// TwinCAT 3 PLC project OEAMTC_WienWest
// ProgramVersion: 3.1.4023.0
// libraries:
//   EfficientIO Communicator, * (EfficientIO)
//   Lynus Energy Basic, * (Lynus AG)
//   Lynus Persistent Data V1, * (Lynus AG)
//   Lynus Standards, * (Lynus AG)
//   Tc2_ModbusRTU, * (Beckhoff Automation GmbH)
//   Tc2_SerialCom, * (Beckhoff Automation GmbH)
//   Tc2_Standard, * (Beckhoff Automation GmbH)
//   Tc2_System, * (Beckhoff Automation GmbH)
//   Tc2_Utilities, * (Beckhoff Automation GmbH)
//   Tc3_Module, * (Beckhoff Automation GmbH)
// project tree:
//   DUTs/ ModbusRTURequest.TcDUT
//   / FastTask.TcTTO, MiddleTask.TcTTO, SlowTask.TcTTO
//   FB/ F_Convert_Reg_to_Real.TcPOU, MODBUS_RTU_v0.TcPOU
//   POUs/ prgComEffIO.TcPOU, prgMain.TcPOU, prgPersistent.TcPOU, prgPV.TcPOU (excluded from build), prgRWEffIO.TcPOU, prgVarEffIO.TcPOU
// real-time tasks:
//   TASK MiddleTask: cycle T#10ms, priority 20, ADS port 350
//   TASK SlowTask: cycle T#20ms, priority 21, ADS port 351
//   TASK FastTask: cycle T#5ms, priority 19, ADS port 352
// I/O:
//   DEVICE Device 1 (Beckhoff CCAT)
//   DEVICE Device 2 (CX-BK)
//     Box 1 (CX-BK)
// variable links:
//   OEAMTC_WienWest/OEAMTC_WienWest Instance <-> Device 2 (CX-BK)/Box 1 (CX-BK)
//     FastTask Inputs/MODBUS_RTU_v0.fbModbusRtuMaster_KL6x22B.InData/D <-> Term 2 (KL6041)/Channel 1/Data In 0
//     FastTask Inputs/MODBUS_RTU_v0.fbModbusRtuMaster_KL6x22B.InData/D @bit {8..168 step 8} <-> Term 2 (KL6041)/Channel 1/Data In {1..21}  (21 links)
//     FastTask Inputs/MODBUS_RTU_v0.fbModbusRtuMaster_KL6x22B.InData/Status <-> Term 2 (KL6041)/Channel 1/State
//     FastTask Inputs/prgMain.fbKBusState.uiKBusState_OUT <-> Inputs/State
//     FastTask Outputs/MODBUS_RTU_v0.fbModbusRtuMaster_KL6x22B.OutData/Ctrl <-> Term 2 (KL6041)/Channel 1/Ctrl
//     FastTask Outputs/MODBUS_RTU_v0.fbModbusRtuMaster_KL6x22B.OutData/D <-> Term 2 (KL6041)/Channel 1/Data Out 0
//     FastTask Outputs/MODBUS_RTU_v0.fbModbusRtuMaster_KL6x22B.OutData/D @bit {8..168 step 8} <-> Term 2 (KL6041)/Channel 1/Data Out {1..21}  (21 links)

CONFIGURATION OEAMTC_WienWest
    RESOURCE PLC ON TwinCAT3
        TASK FastTask(INTERVAL := T#5ms, PRIORITY := 19);
        TASK MiddleTask(INTERVAL := T#10ms, PRIORITY := 20);
        TASK SlowTask(INTERVAL := T#20ms, PRIORITY := 21);
        PROGRAM prgRWEffIO WITH FastTask : prgRWEffIO;
        PROGRAM prgVarEffIO WITH FastTask : prgVarEffIO;
        PROGRAM prgMain WITH FastTask : prgMain;
        PROGRAM prgPersistent WITH MiddleTask : prgPersistent;
        PROGRAM prgComEffIO WITH SlowTask : prgComEffIO;
    END_RESOURCE
END_CONFIGURATION

// ---- DUTs/ModbusRTURequest.TcDUT
TYPE ModbusRTURequest :
STRUCT
	byteClientSlaveID	:BYTE;
	uintStartAddress	:UINT;
	uintNoOfWords		:UINT;
	mError				:BOOL;
	udintErrorID		:MODBUS_ERRORS;
	udintBytesReceived	:UDINT;
	timerErrorTimer		:TON;
	timerOKTimer		:TON;
	wArrayReceiveBuffer	:ARRAY[0..130] OF WORD;
	udintReceiveBufferAddress	:UDINT;
	strErrorMessage		:STRING(50);
	udintCommErrorCounter		:UDINT;
	udintCommSuccessCounter		:UDINT;
	timeTimeForRequest	:TIME;
	mRequestActive		:BOOL;
	intDeviceClass		:INT;
	intDeviceNumber		:INT;
END_STRUCT
END_TYPE

// ---- POUs/prgRWEffIO.TcPOU
PROGRAM prgRWEffIO
VAR
	fbRW1		: FB_ReadWrite_V2;
END_VAR

fbRW1(	eUploadType := 4,
		bBusy=> , 
		bError=> , 
		udiErrorCodeOut=> , 
		eErrorReadWrite_Out=> );

END_PROGRAM

// ---- POUs/prgVarEffIO.TcPOU
PROGRAM prgVarEffIO
VAR
	fbVar			: FB_VarInfo;
END_VAR

fbVar(
	bReadInfo:= , 
	eTMCFile:= eSelectTMCFile.eDontUseTMCFile, 
	eSavePositionTMCFile:= eSavePositionOnPLC.ePostionHardDisk, 
	udiCounterFoundVariables=> , 
	bError=> , 
	bBusy=> , 
	byProgress=> , 
	udiErrorCodeOut=> , 
	eErrorVarInfo_Out=> , 
	sVarWithError=> );

END_PROGRAM

// ---- POUs/prgMain.TcPOU
PROGRAM prgMain
VAR
	lrRealPower1_kW			: LREAL;						//{#lynus.ag#()}
	lrReactivePower1_kVar	: LREAL;						//{#lynus.ag#()}
	lrApparentPower1_VA		: LREAL;						//{#lynus.ag#()}
	rVoltage1_L1N_V			: REAL;							//{#lynus.ag#()}
	rVoltage1_L2N_V			: REAL;							//{#lynus.ag#()}
	rVoltage1_L3N_V			: REAL;							//{#lynus.ag#()}
	rVoltage1_L12_V			: REAL;							//{#lynus.ag#()}
	rVoltage1_L23_V			: REAL;							//{#lynus.ag#()}
	rVoltage1_L31_V			: REAL;							//{#lynus.ag#()}
	rCurrent1_L1_A			: REAL;							//{#lynus.ag#()}
	rCurrent1_L2_A			: REAL;							//{#lynus.ag#()}
	rCurrent1_L3_A			: REAL;							//{#lynus.ag#()}

	lrRealPower2_kW			: LREAL;						//{#lynus.ag#()}
	lrReactivePower2_kVar	: LREAL;						//{#lynus.ag#()}
	lrApparentPower2_VA		: LREAL;						//{#lynus.ag#()}
	rVoltage2_L1N_V			: REAL;							//{#lynus.ag#()}
	rVoltage2_L2N_V			: REAL;							//{#lynus.ag#()}
	rVoltage2_L3N_V			: REAL;							//{#lynus.ag#()}
	rVoltage2_L12_V			: REAL;							//{#lynus.ag#()}
	rVoltage2_L23_V			: REAL;							//{#lynus.ag#()}
	rVoltage2_L31_V			: REAL;							//{#lynus.ag#()}
	rCurrent2_L1_A			: REAL;							//{#lynus.ag#()}
	rCurrent2_L2_A			: REAL;							//{#lynus.ag#()}
	rCurrent2_L3_A			: REAL;							//{#lynus.ag#()}
	fbConvertEnergyRegister		: FB_CV_WORD_TO_DWORD;								//Convert function
	fbGrid1Counter				: FB_EnergyCounter;
	fbGrid2Counter				: FB_EnergyCounter;
	fbKBusState					: FB_K_Bus_State;
	
END_VAR

VAR PERSISTENT
	lrCounterGrid1Prod		: LREAL;								//{#lynus.ag#()}
	lrCounterGrid1Cons		: LREAL;								//{#lynus.ag#()}
	lrCounterGrid2Prod		: LREAL;								//{#lynus.ag#()}
	lrCounterGrid2Cons		: LREAL;								//{#lynus.ag#()}
END_VAR

MODBUS_RTU_v0();


(* Device 1 KBR Multimess NHSV 2*)

rVoltage2_L1N_V :=	rVoltage2_L12_V/(SQRT(3));		// don't understand why I can't get the first voltage from reg 0
rVoltage2_L2N_V := 	F_Convert_Reg_to_Real(	word_in1:=MODBUS_RTU_v0.structArrayModbusRTU[1].wArrayReceiveBuffer[1],
											word_in2:=MODBUS_RTU_v0.structArrayModbusRTU[1].wArrayReceiveBuffer[2]);
rVoltage2_L3N_V := 	F_Convert_Reg_to_Real(	word_in1:=MODBUS_RTU_v0.structArrayModbusRTU[1].wArrayReceiveBuffer[3],
											word_in2:=MODBUS_RTU_v0.structArrayModbusRTU[1].wArrayReceiveBuffer[4]);				
rVoltage2_L12_V := 	F_Convert_Reg_to_Real(	word_in1:=MODBUS_RTU_v0.structArrayModbusRTU[1].wArrayReceiveBuffer[5],
											word_in2:=MODBUS_RTU_v0.structArrayModbusRTU[1].wArrayReceiveBuffer[6]);
rVoltage2_L23_V := 	F_Convert_Reg_to_Real(	word_in1:=MODBUS_RTU_v0.structArrayModbusRTU[1].wArrayReceiveBuffer[7],
											word_in2:=MODBUS_RTU_v0.structArrayModbusRTU[1].wArrayReceiveBuffer[8]);
rVoltage2_L31_V := 	F_Convert_Reg_to_Real(	word_in1:=MODBUS_RTU_v0.structArrayModbusRTU[1].wArrayReceiveBuffer[9],
											word_in2:=MODBUS_RTU_v0.structArrayModbusRTU[1].wArrayReceiveBuffer[10]);
rCurrent2_L1_A := 	F_Convert_Reg_to_Real(	word_in1:=MODBUS_RTU_v0.structArrayModbusRTU[1].wArrayReceiveBuffer[11],
											word_in2:=MODBUS_RTU_v0.structArrayModbusRTU[1].wArrayReceiveBuffer[12]);
rCurrent2_L2_A := 	F_Convert_Reg_to_Real(	word_in1:=MODBUS_RTU_v0.structArrayModbusRTU[1].wArrayReceiveBuffer[13],
											word_in2:=MODBUS_RTU_v0.structArrayModbusRTU[1].wArrayReceiveBuffer[14]);
rCurrent2_L3_A := 	F_Convert_Reg_to_Real(	word_in1:=MODBUS_RTU_v0.structArrayModbusRTU[1].wArrayReceiveBuffer[15],
											word_in2:=MODBUS_RTU_v0.structArrayModbusRTU[1].wArrayReceiveBuffer[16]);
lrApparentPower2_VA := 	(F_Convert_Reg_to_Real(	word_in1:=MODBUS_RTU_v0.structArrayModbusRTU[1].wArrayReceiveBuffer[23],
												word_in2:=MODBUS_RTU_v0.structArrayModbusRTU[1].wArrayReceiveBuffer[24])+
						F_Convert_Reg_to_Real(	word_in1:=MODBUS_RTU_v0.structArrayModbusRTU[1].wArrayReceiveBuffer[25],
												word_in2:=MODBUS_RTU_v0.structArrayModbusRTU[1].wArrayReceiveBuffer[26])+
						F_Convert_Reg_to_Real(	word_in1:=MODBUS_RTU_v0.structArrayModbusRTU[1].wArrayReceiveBuffer[27],
												word_in2:=MODBUS_RTU_v0.structArrayModbusRTU[1].wArrayReceiveBuffer[28]))/1000;
lrRealPower2_kW		:= 	(F_Convert_Reg_to_Real(	word_in1:=MODBUS_RTU_v0.structArrayModbusRTU[1].wArrayReceiveBuffer[29],
												word_in2:=MODBUS_RTU_v0.structArrayModbusRTU[1].wArrayReceiveBuffer[30])+
						F_Convert_Reg_to_Real(	word_in1:=MODBUS_RTU_v0.structArrayModbusRTU[1].wArrayReceiveBuffer[31],
												word_in2:=MODBUS_RTU_v0.structArrayModbusRTU[1].wArrayReceiveBuffer[32])+
						F_Convert_Reg_to_Real(	word_in1:=MODBUS_RTU_v0.structArrayModbusRTU[1].wArrayReceiveBuffer[33],
												word_in2:=MODBUS_RTU_v0.structArrayModbusRTU[1].wArrayReceiveBuffer[34]))/1000;											
lrReactivePower2_kVar:= (F_Convert_Reg_to_Real(	word_in1:=MODBUS_RTU_v0.structArrayModbusRTU[1].wArrayReceiveBuffer[35],
												word_in2:=MODBUS_RTU_v0.structArrayModbusRTU[1].wArrayReceiveBuffer[36])+
						F_Convert_Reg_to_Real(	word_in1:=MODBUS_RTU_v0.structArrayModbusRTU[1].wArrayReceiveBuffer[37],
												word_in2:=MODBUS_RTU_v0.structArrayModbusRTU[1].wArrayReceiveBuffer[38])+
						F_Convert_Reg_to_Real(	word_in1:=MODBUS_RTU_v0.structArrayModbusRTU[1].wArrayReceiveBuffer[39],
												word_in2:=MODBUS_RTU_v0.structArrayModbusRTU[1].wArrayReceiveBuffer[40]))/1000;											

// EnergyCounter
fbGrid2Counter(
	byActiveTariff:= 1, 
	lrPowerInput:= lrRealPower2_kW, 
	lrTotalCounterEnergy_Consumption=> , 
	lrTotalCounterEnergy_Production=> , 
	lrCounterEnergyT1_Consumption=> , 
	lrCounterEnergyT2_Consumption=> , 
	lrCounterEnergyT1_Production=> , 
	lrCounterEnergyT2_Production=> );
	
IF fbGrid2Counter.lrTotalCounterEnergy_Production > lrCounterGrid2Prod THEN  	
	lrCounterGrid2Prod := fbGrid2Counter.lrTotalCounterEnergy_Production;
END_IF	
IF fbGrid2Counter.lrTotalCounterEnergy_Consumption > lrCounterGrid2Cons THEN  	
	lrCounterGrid2Cons := fbGrid2Counter.lrTotalCounterEnergy_Consumption;
END_IF	

//(* Device 2 Celsa TNM96 NHSV 1 *)

rVoltage1_L1N_V :=	rVoltage1_L12_V/(SQRT(3));		// don't understand why I can't get the first voltage from reg 0
rVoltage1_L2N_V := 	F_Convert_Reg_to_Real(	word_in1:=MODBUS_RTU_v0.structArrayModbusRTU[2].wArrayReceiveBuffer[1],
											word_in2:=MODBUS_RTU_v0.structArrayModbusRTU[2].wArrayReceiveBuffer[2]);
rVoltage1_L3N_V := 	F_Convert_Reg_to_Real(	word_in1:=MODBUS_RTU_v0.structArrayModbusRTU[2].wArrayReceiveBuffer[3],
											word_in2:=MODBUS_RTU_v0.structArrayModbusRTU[2].wArrayReceiveBuffer[4]);				
rVoltage1_L12_V := 	F_Convert_Reg_to_Real(	word_in1:=MODBUS_RTU_v0.structArrayModbusRTU[2].wArrayReceiveBuffer[5],
											word_in2:=MODBUS_RTU_v0.structArrayModbusRTU[2].wArrayReceiveBuffer[6]);
rVoltage1_L23_V := 	F_Convert_Reg_to_Real(	word_in1:=MODBUS_RTU_v0.structArrayModbusRTU[2].wArrayReceiveBuffer[7],
											word_in2:=MODBUS_RTU_v0.structArrayModbusRTU[2].wArrayReceiveBuffer[8]);
rVoltage1_L31_V := 	F_Convert_Reg_to_Real(	word_in1:=MODBUS_RTU_v0.structArrayModbusRTU[2].wArrayReceiveBuffer[9],
											word_in2:=MODBUS_RTU_v0.structArrayModbusRTU[2].wArrayReceiveBuffer[10]);
rCurrent1_L1_A := 	F_Convert_Reg_to_Real(	word_in1:=MODBUS_RTU_v0.structArrayModbusRTU[2].wArrayReceiveBuffer[11],
											word_in2:=MODBUS_RTU_v0.structArrayModbusRTU[2].wArrayReceiveBuffer[12]);
rCurrent1_L2_A := 	F_Convert_Reg_to_Real(	word_in1:=MODBUS_RTU_v0.structArrayModbusRTU[2].wArrayReceiveBuffer[13],
											word_in2:=MODBUS_RTU_v0.structArrayModbusRTU[2].wArrayReceiveBuffer[14]);
rCurrent1_L3_A := 	F_Convert_Reg_to_Real(	word_in1:=MODBUS_RTU_v0.structArrayModbusRTU[2].wArrayReceiveBuffer[15],
											word_in2:=MODBUS_RTU_v0.structArrayModbusRTU[2].wArrayReceiveBuffer[16]);
lrRealPower1_kW		:= 	(F_Convert_Reg_to_Real(	word_in1:=MODBUS_RTU_v0.structArrayModbusRTU[2].wArrayReceiveBuffer[23],
												word_in2:=MODBUS_RTU_v0.structArrayModbusRTU[2].wArrayReceiveBuffer[24]))/1000;											
											
lrApparentPower1_VA := 	(F_Convert_Reg_to_Real(	word_in1:=MODBUS_RTU_v0.structArrayModbusRTU[2].wArrayReceiveBuffer[31],
												word_in2:=MODBUS_RTU_v0.structArrayModbusRTU[2].wArrayReceiveBuffer[32]))/1000;
												
lrReactivePower1_kVar:= (F_Convert_Reg_to_Real(	word_in1:=MODBUS_RTU_v0.structArrayModbusRTU[2].wArrayReceiveBuffer[39],
												word_in2:=MODBUS_RTU_v0.structArrayModbusRTU[2].wArrayReceiveBuffer[40]))/1000;																		

												
												// EnergyCounter
fbGrid1Counter(
	byActiveTariff:= 1, 
	lrPowerInput:= lrRealPower1_kW, 
	lrTotalCounterEnergy_Consumption=> , 
	lrTotalCounterEnergy_Production=> , 
	lrCounterEnergyT1_Consumption=> , 
	lrCounterEnergyT2_Consumption=> , 
	lrCounterEnergyT1_Production=> , 
	lrCounterEnergyT2_Production=> );
	
IF fbGrid1Counter.lrTotalCounterEnergy_Production > lrCounterGrid1Prod THEN  	
	lrCounterGrid1Prod := fbGrid1Counter.lrTotalCounterEnergy_Production;
END_IF	
IF fbGrid1Counter.lrTotalCounterEnergy_Consumption > lrCounterGrid1Cons THEN  	
	lrCounterGrid1Cons := fbGrid1Counter.lrTotalCounterEnergy_Consumption;
END_IF	



// kBus reset

fbKBusState(	uiKBusState_OUT=> , 
				b_Kbus_notOk=> , 
				word_ErrorCount=> );

END_PROGRAM

// ---- FB/MODBUS_RTU_v0.TcPOU
PROGRAM MODBUS_RTU_v0

VAR_INPUT

END_VAR
VAR_OUTPUT
	dword_MB_Error		:ARRAY[1..3] OF DWORD;
END_VAR
VAR
	fbModbusRtuMaster_KL6x22B: ModbusRtuMaster_KL6x22B;
	fbConfigKL6041 : KL6Configuration;
	uintPollOrderCount: UINT;
	mBusy: BOOL;
	mError: BOOL;
	mStart: BOOL;
	udintMemoryDestAddress: UDINT;
	udintBytesReceived: UDINT;
	intState: INT:=0;
	timerT1: TON;
	timeWaitT1: TIME:=T#500MS;
	timeWaitT2: TIME:=T#500MS;
	timeNoRxTimeout:	TIME:=T#2S;
	timerT2: TON;

	fb_F_TRIG1: F_TRIG;
	timerTimeout: TON;
	mError_Rx: BOOL;
	udintErrorID: MODBUS_ERRORS;
	byteClientSlaveID: BYTE;
	uintNoOfWords: UINT;
	uintStartAddress: UINT;
	dw_Mask: DWORD;
	dw_Mask_Not: DWORD;
	uint_TestPollOrder: UINT;
	mTestMode: BOOL;
	mInit_Done: BOOL;
	
	structArrayModbusRTU	:ARRAY[1..60] OF ModbusRTURequest;
	uintMaxModbusRTUOrders: UINT;
	mExecute: BOOL;
	int_Handshake: INT:=1;
	mode: ComSerialLineMode_t:=2;
END_VAR

(*
The function block "ModbusRtuMaster_KL6x22B" has 22 bytes where it communicates with the plc
software. These 22 bytes have to be assigned to the hardware device (for example KL/EL6021) in the
system manager plus the control and status byte.
If devices with less then 22 bytes are used, the other function blocks have to be used (for 5 bytes for example).
*)

(*
IF fbModbusRtuMaster_KL6x22B.MBmaster.TimeoutTON.Q=TRUE AND mTimeOUT_Qold=FALSE THEN mTimeOUT_Q_Rising; END_IF
mTimeOUT_Qold:=fbModbusRtuMaster_KL6x22B.MBmaster.TimeoutTON.Q;
*)

fb_F_TRIG1(CLK:=mBusy);

CASE intState OF

0: 	(* reset the start bit *)
	mStart:=FALSE;
	IF mInit_Done AND NOT fbConfigKL6041.Busy THEN 
		intState:=10;
		mExecute:=FALSE;		
	ELSE
		INIT();
		mExecute:=TRUE;		// necessary to write the communication parameters to the KL terminal. only necessary once if the terminal is brand new
	END_IF
10:
	(* set next poll order *)
	uintPollOrderCount:=uintPollOrderCount+1; (* next slave *)
	WHILE NOT structArrayModbusRTU[uintPollOrderCount].mRequestActive DO
		uintPollOrderCount:=uintPollOrderCount+1; (* next slave *)
	END_WHILE
	
	(* trouble shooting *)
	IF mTestMode THEN
		uintPollOrderCount:=uint_TestPollOrder; (* next slave *)
	END_IF
	
	IF uintPollOrderCount > uintMaxModbusRTUOrders OR uintPollOrderCount<1 THEN
		uintPollOrderCount:=1;
	END_IF

	udintMemoryDestAddress:=ADR(structArrayModbusRTU[uintPollOrderCount].wArrayReceiveBuffer[0]);
	structArrayModbusRTU[uintPollOrderCount].udintBytesReceived:=0;
	mStart:=TRUE;
	timerTimeout.IN:=TRUE;
	intState:=20;

20: (* wait for busy falling or time out *)
	IF fb_F_TRIG1.Q OR timerTimeout.Q THEN

		(* check answer time *)
		structArrayModbusRTU[uintPollOrderCount].timeTimeForRequest:=timerTimeout.ET;

		(* reset timer *)
		timerTimeout.IN:=FALSE;

		(* reset start bit *)
		mStart:=FALSE;

		(* save number of bytes received *)
		structArrayModbusRTU[uintPollOrderCount].udintBytesReceived:=udintBytesReceived;
		udintBytesReceived:=0;

		(* Error Detection *)
		IF timerTimeout.Q THEN
			mError_Rx:=TRUE;
			structArrayModbusRTU[uintPollOrderCount].udintErrorID:=9998;
			structArrayModbusRTU[uintPollOrderCount].strErrorMessage:='Timeout';
		ELSIF structArrayModbusRTU[uintPollOrderCount].udintBytesReceived=0 AND structArrayModbusRTU[uintPollOrderCount].uintNoOfWords>0 THEN
			mError_Rx:=TRUE;
			structArrayModbusRTU[uintPollOrderCount].udintErrorID:=9999;
			structArrayModbusRTU[uintPollOrderCount].strErrorMessage:='0 bytes received';
		ELSIF fbModbusRtuMaster_KL6x22B.Error THEN
			mError_Rx:=TRUE;
			structArrayModbusRTU[uintPollOrderCount].udintErrorID:=udintErrorID;
//			structArrayModbusRTU[uintPollOrderCount].strErrorMessage:=F_ADSERRORTEXT(structArrayModbusRTU[uintPollOrderCount].udintErrorID);
		ELSE
			mError_Rx:=FALSE;
			structArrayModbusRTU[uintPollOrderCount].udintErrorID:=0;
			structArrayModbusRTU[uintPollOrderCount].strErrorMessage:='';
		END_IF


		IF mError_Rx THEN
			structArrayModbusRTU[uintPollOrderCount].udintCommErrorCounter:=structArrayModbusRTU[uintPollOrderCount].udintCommErrorCounter+1;
		ELSIF structArrayModbusRTU[uintPollOrderCount].udintBytesReceived>0 THEN (* Rev 3 *)
			structArrayModbusRTU[uintPollOrderCount].udintCommSuccessCounter:=structArrayModbusRTU[uintPollOrderCount].udintCommSuccessCounter+1;
		END_IF

		structArrayModbusRTU[uintPollOrderCount].timerOKTimer.IN:=NOT mError_Rx;
		structArrayModbusRTU[uintPollOrderCount].timerErrorTimer.IN:=mError_Rx;

		dw_Mask:=1;
		dw_Mask:=SHL(dw_Mask,(structArrayModbusRTU[uintPollOrderCount].intDeviceNumber));
		dw_Mask_Not:=NOT dw_Mask;
		
		IF structArrayModbusRTU[uintPollOrderCount].timerErrorTimer.Q THEN
			structArrayModbusRTU[uintPollOrderCount].mError:=TRUE;
			IF structArrayModbusRTU[uintPollOrderCount].intDeviceClass>=1 AND structArrayModbusRTU[uintPollOrderCount].intDeviceClass<=3 THEN
				dword_MB_Error[structArrayModbusRTU[uintPollOrderCount].intDeviceClass]:=dword_MB_Error[structArrayModbusRTU[uintPollOrderCount].intDeviceClass] OR dw_Mask;
			END_IF
		END_IF

		IF structArrayModbusRTU[uintPollOrderCount].timerOKTimer.Q THEN
			structArrayModbusRTU[uintPollOrderCount].mError:=FALSE;
			IF structArrayModbusRTU[uintPollOrderCount].intDeviceClass>=1 AND structArrayModbusRTU[uintPollOrderCount].intDeviceClass<=3 THEN
				dword_MB_Error[structArrayModbusRTU[uintPollOrderCount].intDeviceClass]:=dword_MB_Error[structArrayModbusRTU[uintPollOrderCount].intDeviceClass] AND dw_Mask_Not;
			END_IF
		END_IF

		(* clear buffer *)
		IF mError_Rx THEN
			MEMSET(destAddr:=udintMemoryDestAddress,fillByte:=0,130);
		END_IF

		(* set next state *)
		intState:=30;
	END_IF

30:		(* wait *)
		timerT1(IN:=TRUE);
		IF timerT1.Q THEN
			timerT1(IN:=FALSE);
			intState:=0; (* back to start *)
		END_IF

END_CASE

(* Timer calls *)
structArrayModbusRTU[uintPollOrderCount].timerErrorTimer(PT:=timeNoRxTimeout);
structArrayModbusRTU[uintPollOrderCount].timerOKTimer(PT:=T#2S);
timerT1(PT:=timeWaitT1);
timerT2(PT:=timeWaitT2);
timerTimeout(PT:=timeNoRxTimeout+timeWaitT1);


(* Timers *)
structArrayModbusRTU[uintPollOrderCount].timerErrorTimer.PT:=T#5S;
structArrayModbusRTU[uintPollOrderCount].timerOKTimer.PT:=T#5S;


(*fbModbusRtuMaster_KL6x22B.ReadInputRegs(
*)
fbModbusRtuMaster_KL6x22B.ReadInputRegs(
	UnitID		:=structArrayModbusRTU[uintPollOrderCount].byteClientSlaveID,
	Quantity	:=structArrayModbusRTU[uintPollOrderCount].uintNoOfWords,
	MBAddr		:=structArrayModbusRTU[uintPollOrderCount].uintStartAddress,
	cbLength	:=2*structArrayModbusRTU[uintPollOrderCount].uintNoOfWords,
	pMemoryAddr	:=udintMemoryDestAddress,
	Execute		:=mStart,
	Timeout		:=t#1s,
	BUSY		=>mBusy,
	Error		=>mError,
	ErrorId		=>udintErrorID,
	cbRead		=>udintBytesReceived
);


// necessary for KL6041 to wirte the com settings
fbConfigKL6041(
	Execute 		:= mExecute,
	Mode 			:= mode,
	Baudrate 		:= 19200,
	NoDatabits 		:= 8,
	Parity 			:= 1,
	Stopbits 		:= 1,
	Handshake  		:= int_Handshake,
	ContinousMode 	:= FALSE,
	pComIn 			:= ADR(fbModbusRtuMaster_KL6x22B.InData),
	pComOut 		:= ADR(fbModbusRtuMaster_KL6x22B.OutData),
	SizeComIn 		:= SIZEOF(fbModbusRtuMaster_KL6x22B.InData)
);

ACTION INIT:



(* Device 1 KBR Multimess *)
structArrayModbusRTU[1].byteClientSlaveID:=1;
structArrayModbusRTU[1].uintStartAddress:=1;
structArrayModbusRTU[1].uintNoOfWords:=100;
structArrayModbusRTU[1].mRequestActive:=TRUE;




(* Device 2 Celsa TNM96 *)
structArrayModbusRTU[2].byteClientSlaveID:=31;
structArrayModbusRTU[2].uintStartAddress:=1;
structArrayModbusRTU[2].uintNoOfWords:=80;
structArrayModbusRTU[2].mRequestActive:=TRUE;



uintMaxModbusRTUOrders:=2;
mInit_Done:=TRUE;
END_ACTION

END_PROGRAM

// ---- FB/F_Convert_Reg_to_Real.TcPOU
FUNCTION F_Convert_Reg_to_Real : REAL
VAR_INPUT
	word_in1:WORD;
	word_in2:WORD;
END_VAR
VAR
	word_in	:ARRAY[0..1] OF WORD;
END_VAR

word_in[0]:=word_in1;
word_in[1]:=word_in2;

memcpy(ADR(F_Convert_Reg_to_Real),ADR(word_in),SIZEOF(word_in));

END_FUNCTION

// ---- POUs/prgPersistent.TcPOU
PROGRAM prgPersistent
VAR
	fbUSV		: FB_WritePersistentData_CX81xx;
	fb_Reboot: NT_Reboot;
	mReboot: BOOL:=FALSE;
END_VAR

fbUSV(
	eSaveModeData:= eUSVSaveMode.eSaveWhenPowerfail, 
	bLoadPersistentDataOk=> , 
	bPowerFailDetect=> , 
	bError=> , 
	bySaveProcess=> , 
	dwStorageLast24h=> , 
	udiErrorCode=> );
	
	
fb_Reboot( 	Netid 	:= '',
			Delay	:= 2,
			Start	:= mReboot);

END_PROGRAM

// ---- POUs/prgComEffIO.TcPOU
PROGRAM prgComEffIO
VAR
	fbCom			: FB_MqttCommunicator_V2;
END_VAR

fbCom(
	bConnect:= TRUE,
	strAuthKey :='EIO08031879806',
	sUserName:= '90b3d39e-7421-4c3d-851d-5bcf1221f0e6', 
	sUserPassword:= 'f8bcb488-dc42-4c36-ba45-df0dd9149713', 
	eSavePositionCertificate:= eSavePositionOnPLC.ePostionHardDisk,
	time_HeartBeat_sec	:= T#15S, 
	bConnected=> , 
	bError=> , 
	hrErrorCode=> , 
	eConnectionState=> , 
	eErrorMessage_Out=> );

END_PROGRAM

// ---- POUs/prgPV.TcPOU
PROGRAM prgPV
VAR
	fbKBusState		: FB_K_Bus_State;
	fbEM1			: FB_EM_Beckhoff_KL3403;
	lrPowerEM1		: LREAL;							//{#lynus.ag#()}
	lrCounterEM1	: LREAL;							//{#lynus.ag#()}
END_VAR

fbKBusState(uiKBusState_OUT=> );

//Leistung * 2 weil PV Straenge parallel gefuehrt
fbEM1(
	bEnable:= TRUE, 
	bChannel1Invers:= TRUE,
	bChannel2Invers:= TRUE,
	bChannel3Invers:= TRUE,
	uiCurrentTransformerRatioL1:= 600, 
	uiCurrentTransformerRatioL2:= 600, 
	uiCurrentTransformerRatioL3:= 600, 
	uiKBusState_IN:= fbKBusState.uiKBusState_OUT, 
	stDataEMPower=> , 
	stDataEMCounter=> , 
	stDataEMPowerRealTime=> , 
	stDataEMCounterRealTime=> , 
	diNrOfEM_OUT=> );

lrPowerEM1 := fbEM1.stDataEMPower.lrPowerTotal * 2;	
	lrCounterEM1 := fbEM1.stDataEMCounter.lrTotalCounterEnergy_Consumption * 2;

END_PROGRAM
